(* IEC 61131-3 sources: automatic-screwdriver-line/src/DUT, 9 files *)

(* ---- ActionResult.st ---- *)
// Generated from Automatic_ScrewDriver_Line.xml by tools/export_st.py - do not edit.
// The CODESYS project is the source of truth.

{attribute 'qualified_only'}
{attribute 'strict'}
TYPE ActionResult :
(
	Busy := 1,
	Done,
	Failed
);
END_TYPE

(* ---- ErrorCode.st ---- *)
// Generated from Automatic_ScrewDriver_Line.xml by tools/export_st.py - do not edit.
// The CODESYS project is the source of truth.

{attribute 'qualified_only'}
{attribute 'strict'}
TYPE ErrorCode :
(
	NoError := 0,
	EnablementError,
	ScrewNotReleased,
	TargetNotReached,
	SpindleError,
	CobotNotConnected,
	CobotMovementNotReached,
	RtcNotAvailable
);
END_TYPE

(* ---- JobReport.st ---- *)
// Generated from Automatic_ScrewDriver_Line.xml by tools/export_st.py - do not edit.
// The CODESYS project is the source of truth.

TYPE JobReport :
STRUCT
	JobId : UDINT;
	StartedAt : DT;
	FinishedAt : DT;
	ScrewsOk : INT;
	ScrewsFailed : INT;
	FailedScrews : ScrewList;
	Completed : BOOL;   // TRUE = all screws processed, FALSE = aborted by operator
END_STRUCT
END_TYPE

(* ---- JobState.st ---- *)
// Generated from Automatic_ScrewDriver_Line.xml by tools/export_st.py - do not edit.
// The CODESYS project is the source of truth.

{attribute 'qualified_only'}
{attribute 'strict'}
TYPE JobState :
(
	Idle := 1,
	Reset,
	ReadingTargetPosition,
	MovingToTargetPosition,
	MovingToBase,
	MovingZaxisToTool,
	ProcessingTool,
	MovingZaxisToBase,
	Error
);
END_TYPE

(* ---- MoverState.st ---- *)
// Generated from Automatic_ScrewDriver_Line.xml by tools/export_st.py - do not edit.
// The CODESYS project is the source of truth.

{attribute 'qualified_only'}
{attribute 'strict'}
TYPE MoverState :
(
	Idle := 0,
	WaitingEcho,
	Moving,
	WaitingDoneReleased
);
END_TYPE

(* ---- Screw.st ---- *)
// Generated from Automatic_ScrewDriver_Line.xml by tools/export_st.py - do not edit.
// The CODESYS project is the source of truth.

TYPE Screw :
STRUCT
	PositionMm : REAL;   // in mm
	AngleDeg : DINT;   // in °
END_STRUCT
END_TYPE

(* ---- ScrewList.st ---- *)
// Generated from Automatic_ScrewDriver_Line.xml by tools/export_st.py - do not edit.
// The CODESYS project is the source of truth.

TYPE ScrewList : ARRAY[1..5] OF Screw;
END_TYPE

(* ---- IO_Cobot.st ---- *)
// Generated from Automatic_ScrewDriver_Line.xml by tools/export_st.py - do not edit.
// The CODESYS project is the source of truth.

{attribute 'qualified_only'}
VAR_GLOBAL
	Cmd_Enable : BOOL;   // Type Modbus: coil, Address: 18
	Cmd_Start : BOOL;   // Type Modbus: coil, Address: 16
	Cmd_TargetPos01mm : WORD;   // Type Modbus: register, Address: 128, unit 0.1mm (to keep .1mm resolution from Position)
	Sts_Done : BOOL;   // Type Modbus: coil, Address: 17
	Sts_TargetPosEcho01mm : WORD;   // Type Modbus: register, Address: 129
	Sts_Heartbeat : WORD;   // Type Modbus: register, Address: 130
END_VAR

(* ---- Machine_Constants.st ---- *)
// Generated from Automatic_ScrewDriver_Line.xml by tools/export_st.py - do not edit.
// The CODESYS project is the source of truth.

{attribute 'qualified_only'}
VAR_GLOBAL CONSTANT
	TOOL_SPEED : DINT := 60;   // Speed of the spindle in deg/s
	USE_COBOT : BOOL := TRUE;   // If FALSE then the conveyor is used instead
	LOG_COMPONENT_NAME : STRING := 'ScrewDriverLine';
END_VAR
